FUNCTION_BLOCK TcAxisCommand IMPLEMENTS itfAxisCommand
//VAR_INPUT
//END_VAR
//VAR_OUTPUT
//END_VAR
VAR
	_Command        : ST_Command;	
END_VAR

{warning 'Agregar implementación de método'}
METHOD Abort : MC_Error
END_METHOD

{warning 'Agregar implementación de propiedad'}
PROPERTY Active : BOOL
GET
END_GET
SET
END_SET
END_PROPERTY

{warning 'Agregar implementación de propiedad'}
PROPERTY Busy : BOOL
GET
END_GET
SET
END_SET
END_PROPERTY

{warning 'Agregar implementación de propiedad'}
PROPERTY Command : MC_COMMAND_REF
GET
END_GET
SET
END_SET
END_PROPERTY

{warning 'Agregar implementación de propiedad'}
PROPERTY CommandAborted : BOOL
GET
END_GET
SET
END_SET
END_PROPERTY

{warning 'Agregar implementación de propiedad'}
PROPERTY Done : BOOL
GET
Done := _Command.Done;
END_GET
SET
_Command.Done := Done;
END_SET
END_PROPERTY

{warning 'Agregar implementación de propiedad'}
PROPERTY Error : BOOL
GET
END_GET
SET
END_SET
END_PROPERTY

{warning 'Agregar implementación de propiedad'}
PROPERTY ErrorId : MC_Error
GET
END_GET
SET
END_SET
END_PROPERTY

{warning 'Agregar implementación de propiedad'}
PROPERTY ErrorID_Udint : MC_ErrorID_Udint
GET
END_GET
SET
END_SET
END_PROPERTY

{warning 'add method implementation '}
METHOD Update 		: MC_Error
VAR_INPUT
	Position		: REAL;
	Velocity		: REAL;
	EndVelocity		: REAL;
	Acceleration	: REAL;
	Deceleration	: REAL;
	Jerk			: REAL;
END_VAR
END_METHOD

{warning 'Agregar implementación de método'}
METHOD Wait : MC_Error (* This method only makes sense in the IEC 61499 environment*)
VAR_INPUT
	Timeout	: TIME;
	AbortOnTimeout	: BOOL;
END_VAR
END_METHOD

END_FUNCTION_BLOCK

(* stored: Version 1.1.0.1, ProductVersion 3.1.4024.12
   POU TcAxisCommand: Id {f9a234cf-ef1c-447a-9e2d-1effbffa062c}, SpecialFunc None
   Method Abort: Id {73d26a75-d97b-401a-a630-6f3ab69a36cf}
   Property Active: Id {2834e25f-5b3e-4055-afe9-e1993185f6d8}
   Get Get: Id {5bbb5083-2521-40c2-959f-ffc7cba39078}
   Set Set: Id {5b33df63-c8ce-40fb-b482-3df2c70da172}
   Property Busy: Id {43787a43-7e0d-4b0f-aa57-8cd3ab1ccca9}
   Get Get: Id {a8cb3f27-1627-40ca-b1ab-86f859b1d2ba}
   Set Set: Id {c4ae96c8-7a4c-4a84-9302-805151d78bd8}
   Property Command: Id {7808086b-967a-4cb0-bd3a-e905e936e3a0}
   Get Get: Id {4f900402-595a-439f-9844-26753a89063f}
   Set Set: Id {934e4a00-e9e4-45fa-b8f5-dcac3378d6f5}
   Property CommandAborted: Id {e6964c34-bf16-45be-ab21-8609403aba50}
   Get Get: Id {974bc5d9-3ae6-47ef-bea7-2961ee456450}
   Set Set: Id {0eddba56-ca8e-4551-b2fc-024e5608627e}
   Property Done: Id {d2f02cb9-bfb2-4b84-b210-823e2dd8b296}
   Get Get: Id {a0ff7a23-377e-4df0-a72b-976a415c1e4a}
   Set Set: Id {881fcb83-d5c8-49f6-8663-53b559b03418}
   Property Error: Id {02e03d79-3edb-4be1-8fb8-7cd8f35db3f1}
   Get Get: Id {7d87d008-441f-4a2b-b952-69488e3f45c1}
   Set Set: Id {bb5af801-4296-4411-8443-71ea2c27bec7}
   Property ErrorId: Id {7f05c4f9-3947-49b9-8666-ffd17487ffff}
   Get Get: Id {9c32522d-5215-4f7f-bc8a-e1e8a92612af}
   Set Set: Id {6229fd62-686e-42cc-9c5b-69c80eb5be67}
   Property ErrorID_Udint: Id {91cb70b7-d719-4f6f-9019-5c0daf7f443c}
   Get Get: Id {24da3a79-c7d6-4a9d-af9e-a4660d781206}
   Set Set: Id {3ff2d4f7-188a-4ec7-8645-37ce81ef984a}
   Method Update: Id {0d1a4fff-7089-4186-8730-c136d6df7aa7}
   Method Wait: Id {86e00c72-6bcd-465d-9146-52d4ab58d440} *)
